{attribute 'qualified_only'}
{attribute 'strict'}
{attribute 'to_string'}
TYPE eRobPosType :
(
	Absolut := 0,			// Absolute Bewegung bezogen auf Basis-Koordinatensystem
	Relativ := 1			// Relative Bewegung bezogen auf aktuelle Position
);
END_TYPE

(* stored: Version 1.1.0.1
   DUT eRobPosType: Id {5390dc8e-18b4-4104-955f-d9c541ad834e} *)
